TYPE AxisProperties :
STRUCT
	stIdentification			:		ID;
	stHardware					:		Hardware;
	stApplication				:		Application;
	stHoming					:		Homing;
	stOperationLimits			:		OperationLimits;
END_STRUCT
END_TYPE

(* stored: Version 1.1.0.1, ProductVersion 3.1.4024.6
   DUT AxisProperties: Id {3ec430c3-5241-4ad6-bb60-73e53466afd0} *)
